{attribute 'GeneratedUsingTerminal: KL2531-0001'}
{attribute addProperty BoxType "KL2531-0001"}
{attribute addProperty Description ""}
{attribute addProperty Physics ""}
{attribute addProperty Id "Channel_1AT %Q*Channel_0D1929F00"}
{attribute addProperty CRC "1546867592"}
{attribute addProperty Size "0"}
TYPE KL_5C335388 :
STRUCT
	{attribute addProperty Name "Channel_1"}
	Channel_1 : Channel_0D1929F0;
END_STRUCT
END_TYPE

(* stored: Version 1.2.0.0, ProductVersion 3.1.4024.11
   DUT KL_5C335388: Id {38cd0199-d9d6-4684-84f5-0c32fbe0f3cf} *)
